{attribute addProperty BoxType "EL6001-0000-0016"}
{attribute addProperty Id "CtrlAT %Q*Ctrl_BE606B1B445.51Data_OutAT %Q*ARRAY[0 ..21] OF USINT176220"}
{attribute addProperty CRC "1670428157"}
{attribute addProperty SizeInBites "220"}
{attribute addProperty SizeInBytes "27.5"}
TYPE COM_Outputs_7618C603 :
STRUCT
	{attribute addProperty Name "Ctrl"}
	Ctrl AT %Q* : Ctrl_BE606B1B;
	{attribute addProperty Name "Data_Out"}
	Data_Out AT %Q* : ARRAY[0 ..21] OF USINT;
END_STRUCT
END_TYPE

(* stored: Version 1.2.0.0, ProductVersion 3.1.4024.9
   DUT COM_Outputs_7618C603: Id {67a7869f-dcf9-4c5b-9e96-98564bda1227} *)
